SUBAPPLICATION Uebung_003b (* DigitalInput_I1-2-3-4 auf DigitalOutput_Q1-2-3-4 *)
  (* Standard: 61499-2; Description: Copyright (c) 2023 Meisterschulen am Ostbahnhof This program and the accompanying materials are made available under the terms of the Eclipse Public License 2.0 which is available at https://www.eclipse.org/legal/epl-2.0/ SPDX-License-Identifier: EPL-2.0 *)
  (* Version 1.0, 2023-10-23, Franz Höpfinger, Meisterschulen am Ostbahnhof *)
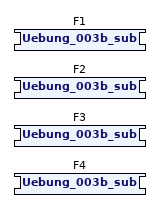
  SUBAPPS
    F1 : Uebung_003b_sub;
    F2 : Uebung_003b_sub;
    F3 : Uebung_003b_sub;
    F4 : Uebung_003b_sub;
  END_SUBAPPS
END_SUBAPPLICATION
